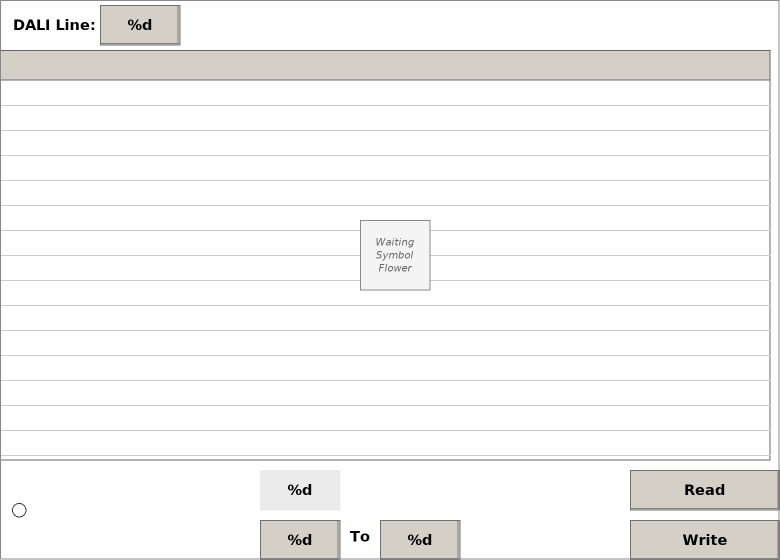
VISUALIZATION Visu_Part103Parameters  // 780x560
    Table (0,50 770x410), data array: DALI_Commissioning.fbPart103Parameters.aParameters
        p1137915858: DALI_Commissioning.fbPart103Parameters.nSelectedAddress
        p3854506369: DALI_Commissioning.fbPart103Parameters.aParameters[INDEX].nOperatingMode
        p1892666644: DALI_Commissioning.fbPart103Parameters.aParameters[INDEX].sInstanceType0
        p338671338: DALI_Commissioning.fbPart103Parameters.aParameters[INDEX].sInstanceType1
        p2170511999: DALI_Commissioning.fbPart103Parameters.aParameters[INDEX].sInstanceType2
        p3723444502: DALI_Commissioning.fbPart103Parameters.aParameters[INDEX].sInstanceType3
        p1218418051: DALI_Commissioning.fbPart103Parameters.aParameters[INDEX].sInstanceType4
        p511219082: IT0 (Generic Input)
        p1755163831: IT1 (PushButton)
        p4092479075: IT2 (Absolute Input)
        p2237128397: IT3 (Occupancy)
        p505689113: IT4 (Light Sensor)
        Columns.Column.[0].Template: OnMouseClick: write the text variable via Default, min 0, max 255, title "Insert Operating Mode 0, 128-255"
    RadioButton (10,460 230x100), variable: DALI_Commissioning.fbPart103Parameters.nAddressRange
        Areas[0]: Text=Single Short Address
        Areas[1]: Text=Short Address Range
    Textfield (260,470 80x40), "%d", text variable: DALI_Commissioning.fbPart103Parameters.nSelectedAddress
    Button (260,520 80x40), "%d", text variable: DALI_Commissioning.fbPart103Parameters.nStartAddress
        OnMouseClick: write the text variable via Default, min 0, max 63, title "Insert Short Address"
    Button (380,520 80x40), "%d", text variable: DALI_Commissioning.fbPart103Parameters.nEndAddress
        OnMouseClick: write the text variable via Default, min 0, max 63, title "Insert Short Address"
    Button (630,470 150x40), "Read"
        OnMouseClick: execute { DALI_Commissioning.fbPart103Parameters.bRead := true; }
    Button (630,520 150x40), "Write"
        OnMouseClick: execute { DALI_Commissioning.fbPart103Parameters.bWrite := true; }
    Textfield (335,521 50x31), "To"
    WaitingSymbolFlower (360,220 70x70), invisible if: DALI_Commissioning.fbPart103Parameters.bHideWaitSymbol
    Group (10,5 170x40)
        Textfield (0,0 110x40), "DALI Line:"
        Button (90,0 80x40), "%d", text variable: GVL_Internal.nDALILine
            OnMouseClick: write the text variable via Default, min 1, max 10, title "Choose line"
END_VISUALIZATION

(* stored: Version 1.1.0.1, ProductVersion 3.1.4024.12
   Visu Visu_Part103Parameters: Id {97a89fd2-a3d7-4a96-a494-e5b809a3cee8} *)
